FUNCTION TryConvert_TIME_TO_REAL : BOOL
VAR_INPUT
	in : TIME;
	out : REFERENCE TO REAL;
END_VAR

out := TIME_TO_REAL(in);
TryConvert_TIME_TO_REAL := TRUE;

END_FUNCTION

(* stored: Version 1.1.0.1, ProductVersion 3.1.4024.12
   POU TryConvert_TIME_TO_REAL: Id {0572ce2b-0a27-4c27-9724-a0146cd6c560}, SpecialFunc None *)
